// TIA Portal V20 export
// export: Created 2025-12-01T14:56:09.1652999Z, ExportSetting None, DisplayName Totally Integrated Automation Portal, DisplayVersion V20 Update 3, DisplayName TIA Portal Openness, DisplayVersion V20 Update 3, DisplayName TIA Portal Version Control Interface, DisplayVersion V20 Update 3, DisplayName STEP 7 Professional, DisplayVersion V20 Update 3, DisplayName STEP 7 Safety, DisplayVersion V20 Update 2, DisplayName WinCC Basic/Comfort/Advanced, DisplayVersion V20 Update 3, DisplayName WinCC Professional, DisplayVersion V20 Update 3, DisplayName WinCC Unified, DisplayVersion V20 Update 3
TYPE "Status_NodosProfinet"
   STRUCT
      Had_Failed { ExternalVisible := 'False'} : Bool;
      Deactivadted { ExternalVisible := 'False'} : Bool;
      Reserved_10 { ExternalVisible := 'False'} : Bool;
      Reseved_11 { ExternalVisible := 'False'} : Bool;
      Reserved_12 { ExternalVisible := 'False'} : Bool;
      Reserved_13 { ExternalVisible := 'False'} : Bool;
      Reserved_14 { ExternalVisible := 'False'} : Bool;
      Reserved_15 { ExternalVisible := 'False'} : Bool;
      OK { ExternalVisible := 'False'} : Bool;
      Maintenance { ExternalVisible := 'False'} : Bool;
      Faulty { ExternalVisible := 'False'} : Bool;
      Failed { ExternalVisible := 'False'} : Bool;
      Was_Deativated { ExternalVisible := 'False'} : Bool;
      DPV1 { ExternalVisible := 'False'} : Bool;
      Was_Under_Maintenace { ExternalVisible := 'False'} : Bool;
      Was_Failed { ExternalVisible := 'False'} : Bool;
   END_STRUCT;
END_TYPE
